PROGRAM MAIN
VAR
	fbModbusMaster 	:		FB_ModbusMaster;
	fbModbusSlave	:		FB_PM2200;
	fbModbusTemp	: 		FB_TDS3000;
	istep			:		UINT;
	bStart			:		BOOL;
	
	arrData			:		ARRAY [0..255] OF BYTE;
END_VAR

CASE istep OF
	0: //Trigger
		IF bStart THEN
			bStart := FALSE;
			istep := 10;
		END_IF
		
	10: //Init
		fbModbusSlave.UnitID := 1;
		fbModbusSlave.FirstCycle();
		fbModbusTemp.UnitID := 2;
		fbModbusTemp.FirstCycle();
		
		fbModbusMaster.FirstCycle();
		fbModbusMaster.Init();
		fbModbusMaster.RegisterSlave(fbModbusSlave);
		fbModbusMaster.RegisterSlave(fbModbusTemp);
		fbModbusMaster.Timeout := 1000;
		istep := 20;
		
	20: //Running
		IF fbModbusMaster.Run() THEN
			istep := 30;
		END_IF
		
	30: //Stopped
		
END_CASE

fbModbusMaster();

END_PROGRAM

(* stored: Version 1.1.0.1, ProductVersion 3.1.4024.12
   POU MAIN: Id {033cb77c-f3de-492f-a9ea-e70326c75ef5}, SpecialFunc None *)
